FUNCTION F_SetHeaderInfo : BOOL
VAR_IN_OUT
	Msg	:ANY;
END_VAR
VAR
END_VAR

END_FUNCTION

(* stored: Version 1.1.0.1, ProductVersion 3.1.4026.17
   POU F_SetHeaderInfo: Id {c0cb69a6-d7df-4110-b29a-d4f544266ffe}, SpecialFunc None *)
